PROGRAM MAIN
VAR
END_VAR

END_PROGRAM

(* stored: Version 1.1.0.1
   POU MAIN: Id {294174a3-fdb4-4db4-8de1-e42c3d8d069a} *)
